// TwinCAT 3 PLC project PLC
// ProgramVersion: 3.1.4024.0
// libraries:
//   Tc2_Standard, * (Beckhoff Automation GmbH)
//   Tc2_System, * (Beckhoff Automation GmbH)
//   Tc3_IPCDiag, * (Beckhoff Automation GmbH)
//   Tc3_Module, * (Beckhoff Automation GmbH)
// project tree:
//   FBs/ FB_GetFullTwinCAT3Version.TcPOU
//   / PlcTask.TcTTO
//   POUs/ MAIN.TcPOU
// real-time tasks:
//   TASK PlcTask: cycle T#10ms, priority 20, ADS port 350

CONFIGURATION PLC
    RESOURCE PLC ON TwinCAT3
        TASK PlcTask(INTERVAL := T#10ms, PRIORITY := 20);
        PROGRAM MAIN WITH PlcTask : MAIN;
    END_RESOURCE
END_CONFIGURATION

// ---- POUs/MAIN.TcPOU
PROGRAM MAIN
VAR
	tonDelay			: TON := (PT := TIME#10S0MS,IN:=TRUE);
	fbGetFullTwinCAT3Version	:FB_GetFullTwinCAT3Version;
END_VAR

tonDelay();
					
fbGetFullTwinCAT3Version(
	cNetId:='' , 
	bStart:=tonDelay.Q , 
	nTCMajor=> , 
	nTCMinor=> , 
	nTCRevision=> , 
	nTCBuild=> , 
	sTCVersion=> );

END_PROGRAM

// ---- FBs/FB_GetFullTwinCAT3Version.TcPOU
FUNCTION_BLOCK FB_GetFullTwinCAT3Version
VAR_INPUT
    cNetId : T_AmsNetID := '';
    bStart : BOOL;
END_VAR
VAR_OUTPUT
    nTCMajor : UINT;
    nTCMinor : UINT;
    nTCRevision : UINT;
    nTCBuild : UINT;
    sTCVersion : STRING;
    hr : HRESULT;
END_VAR
VAR
    rtStart : R_TRIG;
    eState : (Init,
        Idle,
        ReadOnce,
        Error) := Init;

    fbDiagRegister : FB_IPCDiag_Register := (sNetId := cNetId);
    fbDiagRead : FB_IPCDiag_ReadParameter := (sNetId := cNetId);
    nKeyIdx : USINT := 1;
    aParameterKeys : ARRAY[1..cNbrParameters] OF E_IPCDiag_ParameterKey := [E_IPCDiag_ParameterKey.TC_VersionMajor,
        E_IPCDiag_ParameterKey.TC_VersionMinor,
        E_IPCDiag_ParameterKey.TC_VersionRevision,
        E_IPCDiag_ParameterKey.TC_VersionBuild,
        E_IPCDiag_ParameterKey.TC_Version];
END_VAR
VAR CONSTANT
    cNbrParameters : UDINT := 5;
END_VAR

rtStart(CLK := bStart);

CASE eState OF
    Init:
        IF NOT fbDiagRegister.bBusy THEN
            fbDiagRegister(bExecute := TRUE); // need to be executed once
        ELSE
            fbDiagRegister(bExecute := FALSE);
        END_IF

        IF NOT fbDiagRegister.bBusy THEN
            IF fbDiagRegister.bError THEN
                eState := Error;
            ELSE
                eState := Idle;
            END_IF
        END_IF

    Idle:
        IF rtStart.Q THEN
            eState := ReadOnce;
        END_IF

    ReadOnce: // reads every parameter once
        IF NOT fbDiagRead.bBusy THEN
            fbDiagRead(bExecute := TRUE, eParameterKey := aParameterKeys[nKeyIdx], fbRegister := fbDiagRegister);
        ELSE
            fbDiagRead(bExecute := FALSE, fbRegister := fbDiagRegister);
        END_IF

        IF NOT fbDiagRead.bBusy THEN
            IF fbDiagRead.bError THEN
                eState := Error;
            ELSE
                CASE aParameterKeys[nKeyIdx] OF
                    E_IPCDiag_ParameterKey.TC_VersionMajor:
                        hr := fbDiagRead.GetParameter(pBuffer := ADR(nTCMajor), nBufferSize := SIZEOF(nTCMajor));
                    E_IPCDiag_ParameterKey.TC_VersionMinor:
                        hr := fbDiagRead.GetParameter(pBuffer := ADR(nTCMinor), nBufferSize := SIZEOF(nTCMinor));
                    E_IPCDiag_ParameterKey.TC_VersionRevision:
                        hr := fbDiagRead.GetParameter(pBuffer := ADR(nTCRevision), nBufferSize := SIZEOF(nTCRevision));
                    E_IPCDiag_ParameterKey.TC_VersionBuild:
                        hr := fbDiagRead.GetParameter(pBuffer := ADR(nTCBuild), nBufferSize := SIZEOF(nTCBuild));
                    E_IPCDiag_ParameterKey.TC_Version:
                        hr := fbDiagRead.GetParameter(pBuffer := ADR(sTCVersion), nBufferSize := SIZEOF(sTCVersion));
                END_CASE

                IF SUCCEEDED(hr) THEN
                    IF nKeyIdx = cNbrParameters THEN
                        nKeyIdx := 1;
                        eState := Idle;
                    ELSE
                        nKeyIdx := nKeyIdx + 1;
                    END_IF
                ELSE
                    eState := Error;
                END_IF
            END_IF
        END_IF

    Error:
        eState := Idle;

END_CASE

END_FUNCTION_BLOCK
